{attribute 'qualified_only'}
VAR_GLOBAL
	CAN_OUTPUTS AT %Q* : CANTXQUEUESTRUCT_E_32;
	CAN_INPUTS AT %I* : CANRXQUEUESTRUCT_E_32;
END_VAR

(* stored: Version 1.1.0.1
   GVL GVL_PropCAN: Id {674e1022-9ed6-40c0-848d-af13ab364493} *)
